Fanuc KAREL source: kx00018.KL

PROGRAM KX00018
%STACKSIZE=65535
%PRIORITY=65535
%NOLOCKGROUP
VAR
I : INTEGER
J : INTEGER
B : BOOLEAN
F : FILE
S : STRING[80]
P : XYZWPR
-- UNRESOLVED DECLARATIONS (source type spelling not recovered)
-- BA : ARRAY[4] OF TYPE_0x0018 (type_u16=0x2018)
BEGIN
BA[1]=7
-- UNRESOLVED_PC line 13 opcodes [22 9D 33 B1 23] marker_code=19
END KX00018
